// TIA Portal V17 export
// export: Created 2024-10-17T14:16:17.5698332Z, ExportSetting WithDefaults, DisplayName Totally Integrated Automation Portal, DisplayVersion V17 Update 4, DisplayName TIA Portal Openness, DisplayVersion V17 Update 4, DisplayName TIA Portal Version Control Interface, DisplayVersion V17, DisplayName SINAMICS Startdrive Advanced, DisplayVersion V17 Update2, DisplayName SINAMICS Startdrive G130, G150, S120, S150, SINAMICS MV, S210, DisplayVersion V17 Update2, DisplayName SINAMICS Startdrive G110M, G120, G120C, G120D, G120P, G115D, DisplayVersion V17 Update2, DisplayName STEP 7 Professional, DisplayVersion V17 Update 4, DisplayName STEP 7 Safety, DisplayVersion V17, DisplayName WinCC Advanced / Unified PC, DisplayVersion V17 Update 4
TYPE "LPMLV2022_typeDateTime"
TITLE = LPMLV2022_typeDateTime
// Support: tech.team.motioncontrol@siemens.com
// stored: IsFailsafeCompliant false
   STRUCT
      Year { ExternalWritable := 'False'} : Int;
      Month { ExternalWritable := 'False'} : Int;
      Day { ExternalWritable := 'False'} : Int;
      Hour { ExternalWritable := 'False'} : Int;   // (24hr format)
      Minute { ExternalWritable := 'False'} : Int;
      Second { ExternalWritable := 'False'} : Int;
      Millisecond { ExternalWritable := 'False'} : Int;
   END_STRUCT;
END_TYPE
